// TwinCAT 3 PLC project Untitled1
// ProgramVersion: 3.1.4023.0
// libraries:
//   Tc2_Standard, * (Beckhoff Automation GmbH)
//   Tc2_System, * (Beckhoff Automation GmbH)
//   Tc3_Module, * (Beckhoff Automation GmbH)
// project tree:
//   / PlcTask.TcTTO
//   POUs/ MAIN.TcPOU
// real-time tasks:
//   TASK PlcTask: cycle T#10ms, priority 20, ADS port 350

CONFIGURATION Untitled1
    RESOURCE PLC ON TwinCAT3
        TASK PlcTask(INTERVAL := T#10ms, PRIORITY := 20);
        PROGRAM MAIN WITH PlcTask : MAIN;
    END_RESOURCE
END_CONFIGURATION

// ---- POUs/MAIN.TcPOU
PROGRAM MAIN
VAR
	 Delay : TON;
   Count : INT := 0;
	XValueInt : INT;
	YValueInt :INT;
	
END_VAR

Delay(IN:=TRUE, PT:=T#10S);
IF(Delay.Q) THEN
   XValueInt := XValueInt + 1;
   
   
   
END_IF;

Delay(IN:=TRUE);
   
IF (Delay.Q) THEN
	   YValueInt := YValueInt + 3;
END_IF;

END_PROGRAM
